FUNCTION SIGN_R (* this function return true if the real input is negative *)
  (* Standard: 61499-1 *)
  (* Version 1.0, 2025-12-21, franz *)
  PACKAGE OSCAT::Basic::POUs::Mathematical;
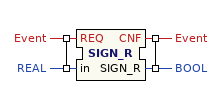
  EVENT_INPUT
    REQ WITH in;
  END_EVENT
  EVENT_OUTPUT
    CNF WITH SIGN_R;
  END_EVENT
  VAR_INPUT
    in : REAL;
  END_VAR
  VAR_OUTPUT
    SIGN_R : BOOL;
  END_VAR
  BODY IN ST:
PACKAGE OSCAT::Basic::POUs::Mathematical;

(* this function return true if the real input is negative *)
FUNCTION SIGN_R : BOOL
VAR_INPUT
	in : REAL;
END_VAR

(*
 * version 1.4	10. mar. 2009 programmer 	hugo tested by		tobias
 *
 * this function return true if the real input is negative
 *)
SIGN_R := in < 0.0;

END_FUNCTION

(* revision history hm 19.1.2007	rev 1.1 changed method of function for better compatibility to
 * other systems
 *
 * hm	1.12.2007	rev 1.2 changed code to improve performance
 *
 * hm	14. jun. 2008	rev 1.3 improved performace
 *
 * hm 10. mar. 2009	rev 1.4 real constants updated to new systax using dot *)
  END_BODY
END_FUNCTION
